PROGRAM CaPart
VAR_INPUT
          iMode                      :INT;
END_VAR

VAR
	fbCaPart: FB_UserMain;
END_VAR

CALL();
ACT();

ACTION ACT:
(********模切小时、天产能**********)
(*
aCaDay_date(
EE:=Q204[7],
);
*)
//运行时间统计
Catimedata(
	Month:= PLC_wMonth, 
	dDay:=PLC_wDay , 
	Hour:=PLC_wHour , 
	Mins:=PLC_wMinute , 
	Second:=PLC_wSecond , 
	Alm:=stSysState.bErrorStop AND NOT bAnDoorALM AND 
             NOT (ProductPar.CaPar.MQ.bWindSelect AND  ProductPar.parFilterAD[13].Out_Value<=ProductPar.CaPar.fDiameterAlarm_L) AND 
             NOT ( NOT ProductPar.CaPar.MQ.bWindSelect AND  ProductPar.parFilterAD[14].Out_Value<=ProductPar.CaPar.fDiameterAlarm_R) , 
	Wait:=(stSysState.iModehmi=2 OR  stSysState.iModehmi=3 )AND (stSysState.bErrorStop OR bAnDoorALM) AND
             NOT (ProductPar.CaPar.MQ.bWindSelect AND  ProductPar.parFilterAD[13].Out_Value<=ProductPar.CaPar.fDiameterAlarm_L) AND 
             NOT ( NOT ProductPar.CaPar.MQ.bWindSelect AND  ProductPar.parFilterAD[14].Out_Value<=ProductPar.CaPar.fDiameterAlarm_R)   , 
	Run:=stSysState.iModehmi=1  , 
	JP_Wait:=(ProductPar.CaPar.MQ.bWindSelect AND  ProductPar.parFilterAD[13].Out_Value<=ProductPar.CaPar.fDiameterAlarm_L) OR ( NOT ProductPar.CaPar.MQ.bWindSelect AND  ProductPar.parFilterAD[14].Out_Value<=ProductPar.CaPar.fDiameterAlarm_R) , 
	Query:=MQQuery , 
	STTimedata=> , 
	date1:=MQdate );
END_ACTION

ACTION CALL:
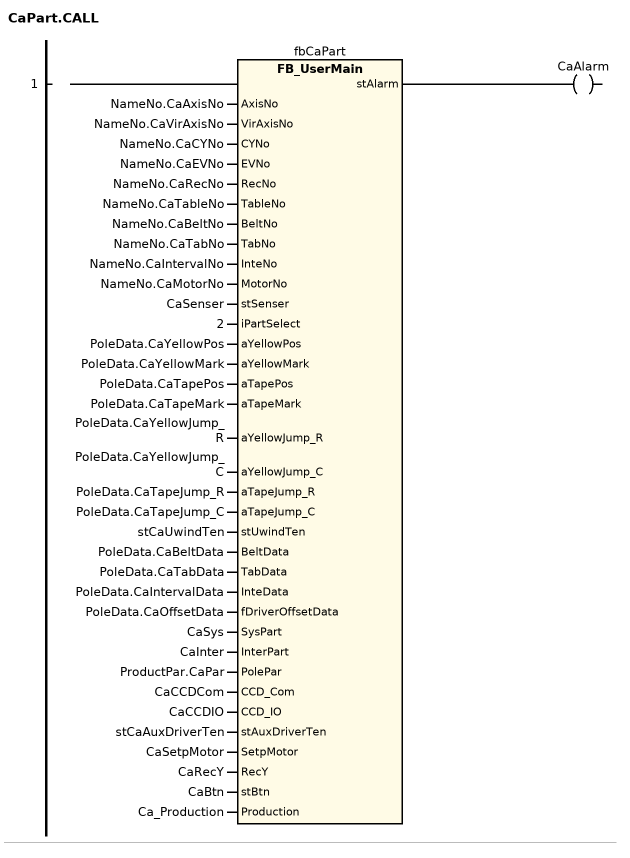
// NETWORK 1
fbCaPart(
    AxisNo := NameNo.CaAxisNo,
    VirAxisNo := NameNo.CaVirAxisNo,
    CYNo := NameNo.CaCYNo,
    EVNo := NameNo.CaEVNo,
    RecNo := NameNo.CaRecNo,
    TableNo := NameNo.CaTableNo,
    BeltNo := NameNo.CaBeltNo,
    TabNo := NameNo.CaTabNo,
    InteNo := NameNo.CaIntervalNo,
    MotorNo := NameNo.CaMotorNo,
    stSenser := CaSenser,
    iPartSelect := 2,
    aYellowPos := PoleData.CaYellowPos,
    aYellowMark := PoleData.CaYellowMark,
    aTapePos := PoleData.CaTapePos,
    aTapeMark := PoleData.CaTapeMark,
    aYellowJump_R := PoleData.CaYellowJump_R,
    aYellowJump_C := PoleData.CaYellowJump_C,
    aTapeJump_R := PoleData.CaTapeJump_R,
    aTapeJump_C := PoleData.CaTapeJump_C,
    stUwindTen := stCaUwindTen,
    BeltData := PoleData.CaBeltData,
    TabData := PoleData.CaTabData,
    InteData := PoleData.CaIntervalData,
    fDriverOffsetData := PoleData.CaOffsetData,
    SysPart := CaSys,
    InterPart := CaInter,
    PolePar := ProductPar.CaPar,
    CCD_Com := CaCCDCom,
    CCD_IO := CaCCDIO,
    stAuxDriverTen := stCaAuxDriverTen,
    SetpMotor := CaSetpMotor,
    RecY := CaRecY,
    stBtn := CaBtn,
    Production := Ca_Production); // FB_UserMain
CaAlarm := fbCaPart.stAlarm;
END_ACTION

END_PROGRAM

(* stored: Version 1.1.0.1, ProductVersion 3.1.4024.12
   POU CaPart: Id {49635e8d-6b0c-4517-8012-ee005f4cf54d}, SpecialFunc None
   Action ACT: Id {f2695612-8fdd-4650-8e67-1ed0feeb4c8e}
   Action CALL: Id {8d802b5b-a0f4-4798-9137-63171d44f9e0} *)
